Staubli VAL3: cycle_getSize.pgx

program cycle_getSize(num& x_nSize[] (dimensions=1), num x_nType (dimensions=1))
  local num l_nID
  local string sName
begin
  //
  // get the size of process list running
  //
  l_nID=0
  call processList:getCycle(sName,l_nID,l_nID,0,x_nType)
  // check if the name is not null
  if sName!=""
    call processList:getSize(x_nSize,x_nType)
  else
    x_nSize=0
  endIf
end
